// TIA Portal V21 export
FUNCTION_BLOCK "Motor Block"   // FB3, LAD
{ S7_Optimized_Access := 'FALSE' }
// stored: AutoNumber false, SetENOAutomatically false
   VAR_INPUT
      Cmd { ExternalVisible := 'False'} : Bool;
      SimulationOn { ExternalVisible := 'False'} : Bool;
      MotorFeedbackInput { ExternalVisible := 'False'} : Bool;
      WaterSensorSelection { ExternalVisible := 'False'} : Bool;
      WaterSensorInput { ExternalVisible := 'False'} : Bool;
      AlwaysTrue : Bool;
      AlwaysFalse : Bool;
      FBCheckDelay { ExternalVisible := 'False'} : Int;
      WSCheckDelay { ExternalVisible := 'False'} : Int;
      secs { ExternalVisible := 'False'} : Bool;
      AlarmAck { ExternalVisible := 'False'} : Bool;
   END_VAR
   VAR_OUTPUT
      Output { ExternalVisible := 'False'} : Bool;
      FeedBackTripAlarm : Bool;
      NoWaterFlowAlarm : Bool;
   END_VAR
   VAR_IN_OUT
      OpFbTrip { ExternalVisible := 'False'} : Bool;
      OpWaterSensorTrip { ExternalVisible := 'False'} : Bool;
      FBCheckActualTime { ExternalVisible := 'False'} : Int;
      WSCheckActualTime { ExternalVisible := 'False'} : Int;
   END_VAR
   VAR_TEMP   // added for the SCL form of the ladder/FBD networks
      _w1 : Bool;
      _w2 : Bool;
   END_VAR
BEGIN

REGION Network 1: OPOn
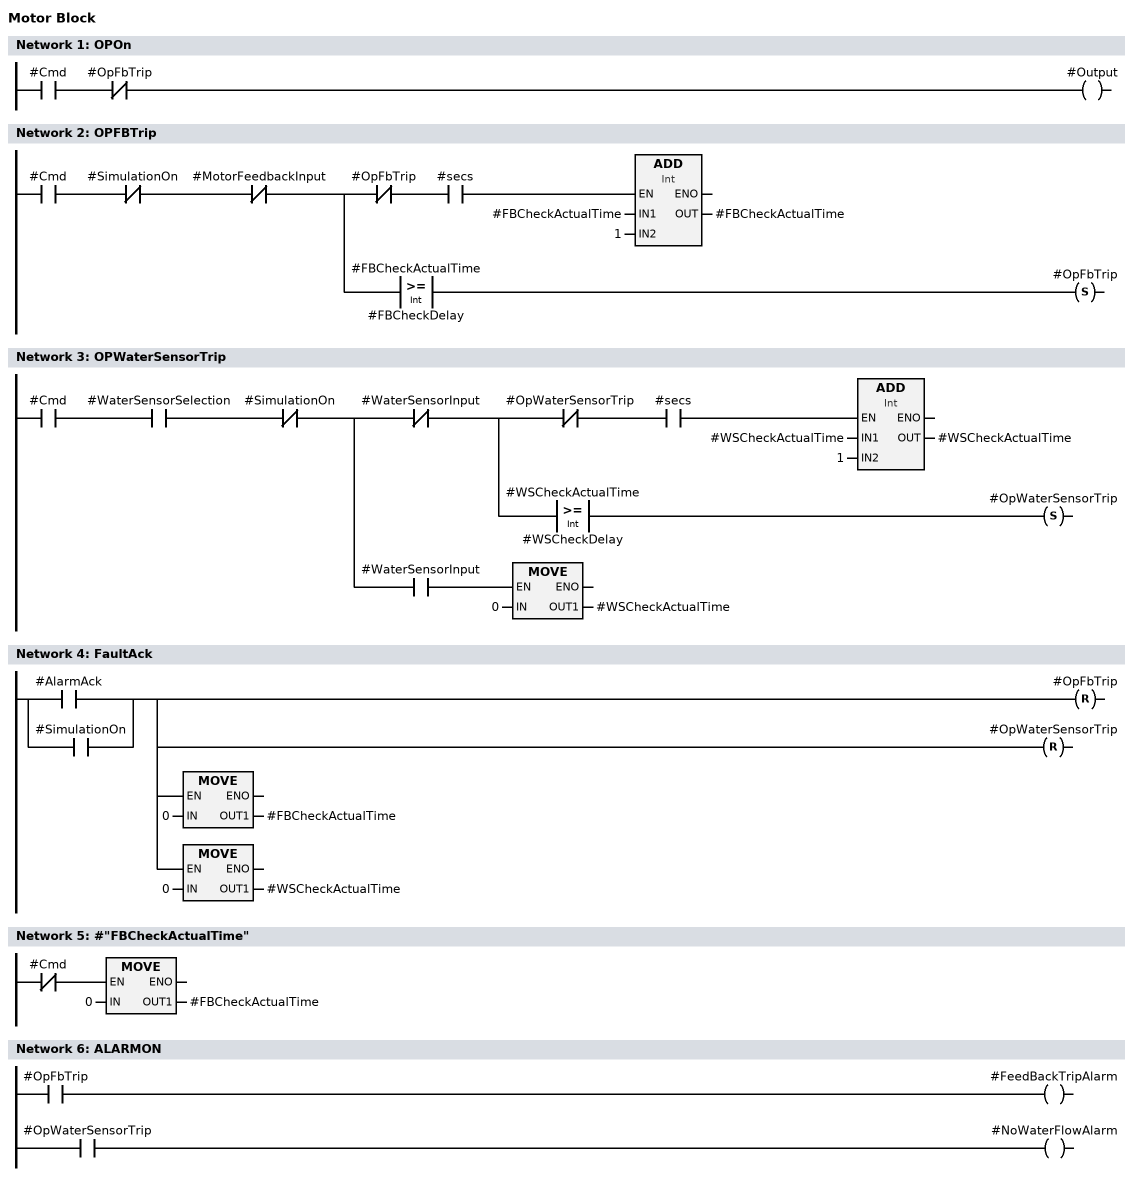
   RUNG wire#powerrail
      Contact( #Cmd )
      I_Contact( #OpFbTrip )
      Coil( #Output )
   END_RUNG
   // the same network as SCL:
   #Output := #Cmd AND NOT #OpFbTrip;
END_REGION

REGION Network 2: OPFBTrip
   RUNG wire#powerrail
      Contact( #Cmd )
      I_Contact( #SimulationOn )
      I_Contact( #MotorFeedbackInput )
      wire#w1
      I_Contact( #OpFbTrip )
      Contact( #secs )
      { S7_Templates := "SrcType := Int"; S7_GenerateENO := "TRUE" } Add(in1 := #FBCheckActualTime, in2 := 1, out => #FBCheckActualTime)
   END_RUNG
   RUNG wire#w1
      { S7_Templates := "SrcType := Int" } GE_Contact(in1 := #FBCheckActualTime, in2 := #FBCheckDelay)
      S_Coil( #OpFbTrip )
   END_RUNG
   // the same network as SCL:
   #_w1 := #Cmd AND NOT #SimulationOn AND NOT #MotorFeedbackInput;
   IF #_w1 AND NOT #OpFbTrip AND #secs THEN #FBCheckActualTime := #FBCheckActualTime + 1; END_IF;
   IF #_w1 AND (#FBCheckActualTime >= #FBCheckDelay) THEN #OpFbTrip := TRUE; END_IF;
END_REGION

REGION Network 3: OPWaterSensorTrip
   RUNG wire#powerrail
      Contact( #Cmd )
      Contact( #WaterSensorSelection )
      I_Contact( #SimulationOn )
      wire#w1
      I_Contact( #WaterSensorInput )
      wire#w2
      I_Contact( #OpWaterSensorTrip )
      Contact( #secs )
      { S7_Templates := "SrcType := Int"; S7_GenerateENO := "TRUE" } Add(in1 := #WSCheckActualTime, in2 := 1, out => #WSCheckActualTime)
   END_RUNG
   RUNG wire#w2
      { S7_Templates := "SrcType := Int" } GE_Contact(in1 := #WSCheckActualTime, in2 := #WSCheckDelay)
      S_Coil( #OpWaterSensorTrip )
   END_RUNG
   RUNG wire#w1
      Contact( #WaterSensorInput )
      { S7_GenerateENO := "TRUE" } Move(in := 0, out1 => #WSCheckActualTime)
   END_RUNG
   // the same network as SCL:
   #_w1 := #Cmd AND #WaterSensorSelection AND NOT #SimulationOn;
   #_w2 := #_w1 AND NOT #WaterSensorInput;
   IF #_w2 AND NOT #OpWaterSensorTrip AND #secs THEN #WSCheckActualTime := #WSCheckActualTime + 1; END_IF;
   IF #_w2 AND (#WSCheckActualTime >= #WSCheckDelay) THEN #OpWaterSensorTrip := TRUE; END_IF;
   IF #_w1 AND #WaterSensorInput THEN #WSCheckActualTime := 0; END_IF;
END_REGION

REGION Network 4: FaultAck
   RUNG wire#powerrail
      Contact( #AlarmAck )
      wire#w1
      R_Coil( #OpFbTrip )
   END_RUNG
   RUNG wire#powerrail
      Contact( #SimulationOn )
   END_RUNG wire#w1
   RUNG wire#w1
      R_Coil( #OpWaterSensorTrip )
   END_RUNG
   RUNG wire#w1
      { S7_GenerateENO := "TRUE" } Move(in := 0, out1 => #FBCheckActualTime)
   END_RUNG
   RUNG wire#w1
      { S7_GenerateENO := "TRUE" } Move(in := 0, out1 => #WSCheckActualTime)
   END_RUNG
   // the same network as SCL:
   IF #AlarmAck OR #SimulationOn THEN
       #OpFbTrip := FALSE;
       #OpWaterSensorTrip := FALSE;
       #FBCheckActualTime := 0;
       #WSCheckActualTime := 0;
   END_IF;
END_REGION

REGION Network 5: #"FBCheckActualTime"
   RUNG wire#powerrail
      I_Contact( #Cmd )
      { S7_GenerateENO := "TRUE" } Move(in := 0, out1 => #FBCheckActualTime)
   END_RUNG
   // the same network as SCL:
   IF NOT #Cmd THEN #FBCheckActualTime := 0; END_IF;
END_REGION

REGION Network 6: ALARMON
   RUNG wire#powerrail
      Contact( #OpFbTrip )
      Coil( #FeedBackTripAlarm )
   END_RUNG
   RUNG wire#powerrail
      Contact( #OpWaterSensorTrip )
      Coil( #NoWaterFlowAlarm )
   END_RUNG
   // the same network as SCL:
   #FeedBackTripAlarm := #OpFbTrip;
   #NoWaterFlowAlarm := #OpWaterSensorTrip;
END_REGION
END_FUNCTION_BLOCK
